{attribute 'linkalways'} 
{attribute 'no_explicit_call' := 'This FB is a CLASS and must be accessed using methods or properties'}
{attribute 'enable_dynamic_creation'}
FUNCTION_BLOCK Node_F_VN_MatchDescriptorsBF EXTENDS VisionNode
VAR
    ipQueryDescriptors : _ITcVnImage;
    ipTrainDescriptors : _ITcVnImage;
    ipMatches : _ITcVnContainer;
    hrPrev : _HRESULT(S_OK);
	hresult : _HRESULT(S_OK);
END_VAR

METHOD PUBLIC  Clone : I_Node
VAR
	pNode : POINTER TO Node_F_VN_MatchDescriptorsBF;
END_VAR
pNode := __NEW(Node_F_VN_MatchDescriptorsBF);
Clone := pNode^;
END_METHOD

METHOD FB_init : BOOL
VAR_INPUT
	bInitRetains : BOOL; // if TRUE, the retain variables are initialized (warm start / cold start)
	bInCopyCode : BOOL;  // if TRUE, the instance afterwards gets moved into the copy code (online change)
END_VAR
AddInput('ipQueryDescriptors', ipQueryDescriptors);
AddInput('ipTrainDescriptors', ipTrainDescriptors);
AddInput('hrPrev', hrPrev);
AddOutput('ipMatches', ipMatches);
AddOutput('hresult',hresult);
END_METHOD

METHOD PROTECTED OnExecute
hresult.Value := F_VN_MatchDescriptorsBF(
	ipQueryDescriptors := ipQueryDescriptors.Value,
    ipTrainDescriptors := ipTrainDescriptors.Value,
    ipMatches := ipMatches.Value,
	hrPrev:= hrPrev.Value);
END_METHOD

METHOD PUBLIC PreExecutionCheck
VAR_INPUT
	Check : I_PreExecutionChecks;
END_VAR
Check.IsTrue(ipQueryDescriptors.IsValid, 'ipQueryDescriptors must contain an image');
Check.IsTrue(ipTrainDescriptors.IsValid, 'ipTrainDescriptors must contain an image');
END_METHOD

END_FUNCTION_BLOCK

(* stored: Version 1.1.0.1, ProductVersion 3.1.4024.13
   POU Node_F_VN_MatchDescriptorsBF: Id {b57fd29d-3639-07b0-3347-7b5b673bcd99}, SpecialFunc None
   Folder Constructor: Id {626d6c8a-449e-010e-2c1c-3db5092f0ac0}
   Method Clone: Id {a04d8b0d-4abb-03e3-3ab5-7f7d3ffb255f}
   Method FB_init: Id {e75ebd13-9186-06f9-2c72-257848ff07f2}
   Method OnExecute: Id {9da14cb4-7fb5-09ea-1efc-8238c2b480a3}
   Method PreExecutionCheck: Id {eca1e3d2-9729-004f-1260-64e98921f911} *)
